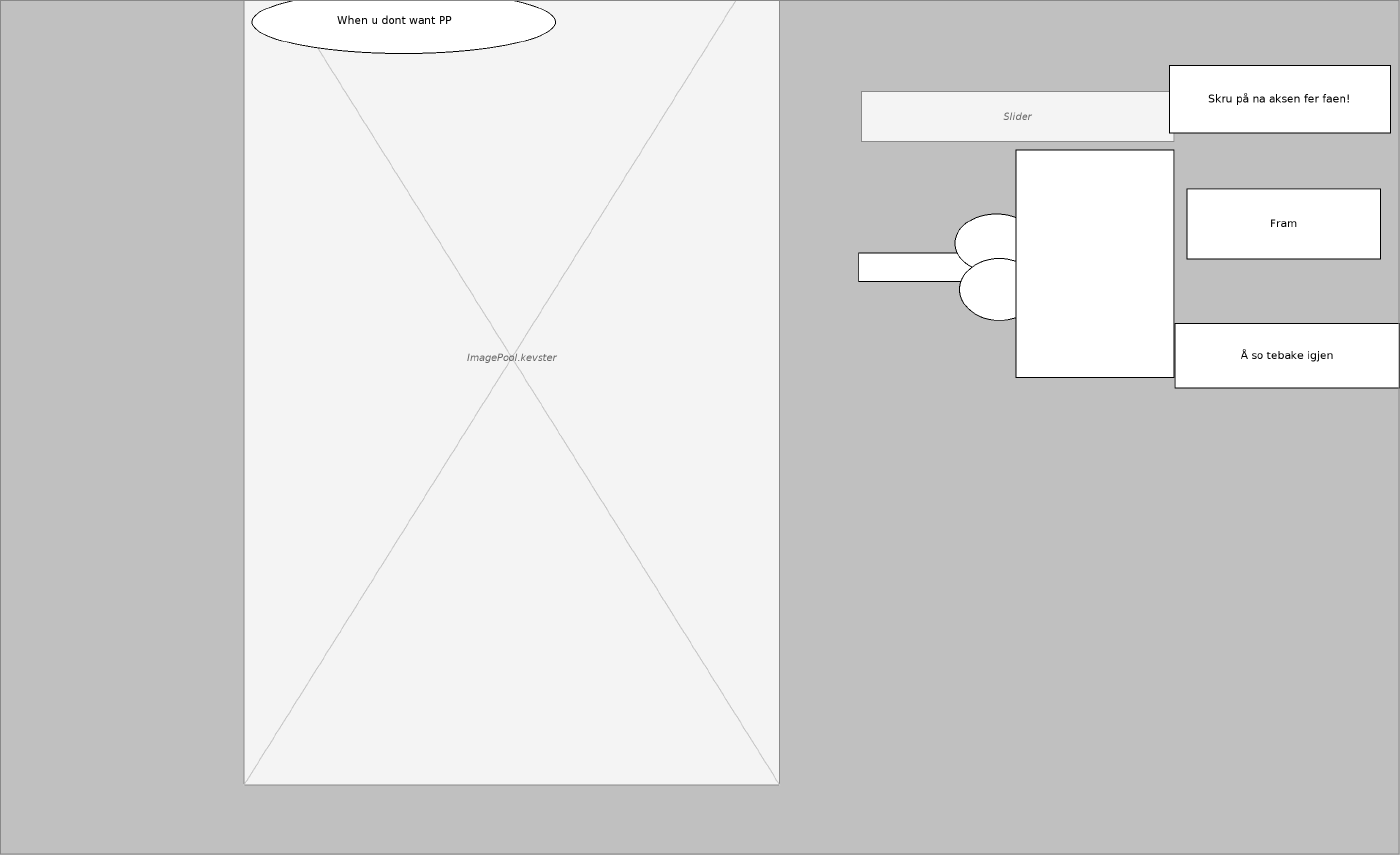
VISUALIZATION Visualization  // 1442x881
    Image (251,-72 552x881), image: ImagePool.kevster
    RoundedRectangle (884,260 312x30)
        p3528305787: -HAVL.actualPosition/10
    Ellipse (983,220 86x61)
    Ellipse (988,266 82x64)
    Slider (887,94 322x52), scale 0..100
    RoundedRectangle (1204,67 228x70), "Skru på na aksen fer faen!", tooltip "Blir brukt fer å skru på aksen!"
        toggle HAVL.enable
    RoundedRectangle (1222,194 200x73), "Fram"
        toggle HAVL.forward
    RoundedRectangle (1210,333 232x67), "Å so tebake igjen"
        toggle HAVL.backwards
    Ellipse (259,-10 313x65)
    Label (331,6 150x30), "When u dont want PP"
    RoundedRectangle (1046,154 163x235)
END_VISUALIZATION

(* stored: Version 1.1.0.1, ProductVersion 3.1.4024.6
   Visu Visualization: Id {80e49fed-d5fc-44d9-a530-ce85c4fb860f} *)
